KUKA KRL data list: A_154.dat

&ACCESS RVP
&REL 89
&PARAM EDITMASK = *
&PARAM TEMPLATE = C:\KRC\Roboter\Template\vorgabe
&PARAM DISKPATH = KRC:\R1\Program\T
DEFDAT  A_154
;FOLD EXTERNAL DECLARATIONS;%{PE}%MKUKATPBASIS,%CEXT,%VCOMMON,%P
;FOLD BASISTECH EXT;%{PE}%MKUKATPBASIS,%CEXT,%VEXT,%P
EXT  BAS (BAS_COMMAND  :IN,REAL  :IN )
DECL INT SUCCESS
;ENDFOLD (BASISTECH EXT)
;FOLD USER EXT;%{E}%MKUKATPUSER,%CEXT,%VEXT,%P
;Make your modifications here

;ENDFOLD (USER EXT)
;ENDFOLD (EXTERNAL DECLARATIONS)


DECL E6POS POS2={X 0.0,Y 0.0,Z 0.0,A 0.0,B 0.0,C 0.0}
DECL FDAT FS2={TOOL_NO 1,BASE_NO 1,IPO_FRAME #BASE,POINT2[] " ",TQ_STATE FALSE}
DECL LDAT LL2={VEL 0.0450000,ACC 100.000,APO_DIST 55.0000,APO_FAC 50.0000,AXIS_VEL 100.000,AXIS_ACC 100.000,ORI_TYP #VAR,CIRC_TYP #BASE,JERK_FAC 50.0000,GEAR_JERK 50.0000,EXAX_IGN 0}
DECL E6POS XP1={X 1765.00,Y -1.00106798E-34,Z 1784.00,A 0.0,B 90.0000,C 3.24968692E-36,S 2,T 34,E1 0.0,E2 0.0,E3 0.0,E4 0.0,E5 0.0,E6 0.0}
DECL FDAT FP1={TOOL_NO 1,BASE_NO 0,IPO_FRAME #BASE,POINT2[] " "}
DECL PDAT PPDAT1={VEL 100.000,ACC 100.000,APO_DIST 100.000,APO_MODE #CPTP,GEAR_JERK 100.000,EXAX_IGN 0}
DECL MODULEPARAM_T LAST_TP_PARAMS={PARAMS[] "Kuka.PointName=P6; Kuka.FrameData.base_no=0; Kuka.FrameData.tool_no=1; Kuka.FrameData.ipo_frame=#BASE; Kuka.isglobalpoint=False; Kuka.MoveDataPtpName=PDAT6; Kuka.MovementDataPdat.apo_mode=#CPTP; Kuka.MovementDataPdat.apo_dist=100; Kuka.MovementData.vel=100; Kuka.MovementData.acc=100; Kuka.MovementData.gear_jerk=100; Kuka.MovementData.exax_ign=0; Kuka.VelocityPtp=100; Kuka.BlendingEnabled=False; Kuka.CurrentCDSetIndex=0          "}
DECL E6POS XP2={X 1765.00,Y -1.00106855E-34,Z 1784.00,A 0.0,B 90.0000,C 3.24968513E-36,S 2,T 34,E1 0.0,E2 0.0,E3 0.0,E4 0.0,E5 0.0,E6 0.0}
DECL FDAT FP2={TOOL_NO 1,BASE_NO 0,IPO_FRAME #BASE,POINT2[] " "}
DECL PDAT PPDAT2={VEL 100.000,ACC 100.000,APO_DIST 100.000,APO_MODE #CPTP,GEAR_JERK 100.000,EXAX_IGN 0}
DECL E6POS XP3={X 1765.00,Y -1.00106752E-34,Z 1784.00,A 0.0,B 90.0000,C 3.24968513E-36,S 2,T 2,E1 0.0,E2 0.0,E3 0.0,E4 0.0,E5 0.0,E6 0.0}
DECL FDAT FP3={TOOL_NO 1,BASE_NO 0,IPO_FRAME #BASE,POINT2[] " "}
DECL PDAT PPDAT3={VEL 100.000,ACC 100.000,APO_DIST 100.000,APO_MODE #CPTP,GEAR_JERK 100.000,EXAX_IGN 0}
DECL E6POS XP4={X 1795.10388,Y 3.17657602E-24,Z 1784.00,A 0.0,B 90.0000,C -1.03118683E-25,S 2,T 43,E1 0.0,E2 0.0,E3 0.0,E4 0.0,E5 0.0,E6 0.0}
DECL FDAT FP4={TOOL_NO 1,BASE_NO 0,IPO_FRAME #BASE,POINT2[] " "}
DECL PDAT PPDAT4={VEL 100.000,ACC 100.000,APO_DIST 100.000,APO_MODE #CPTP,GEAR_JERK 100.000,EXAX_IGN 0}
DECL E6POS XP5={X 1795.10388,Y 0.186128840,Z 1783.99988,A 0.0,B 90.0000458,C -1.50988681E-05,S 2,T 35,E1 0.0,E2 0.0,E3 0.0,E4 0.0,E5 0.0,E6 0.0}
DECL FDAT FP5={TOOL_NO 1,BASE_NO 0,IPO_FRAME #BASE,POINT2[] " "}
DECL PDAT PPDAT5={VEL 100.000,ACC 100.000,APO_DIST 100.000,APO_MODE #CPTP,GEAR_JERK 100.000,EXAX_IGN 0}
DECL E6POS XP6={X 1795.10388,Y 0.588755548,Z 1783.99939,A 0.0,B 90.0001526,C -4.70552841E-05,S 2,T 35,E1 0.0,E2 0.0,E3 0.0,E4 0.0,E5 0.0,E6 0.0}
DECL FDAT FP6={TOOL_NO 1,BASE_NO 0,IPO_FRAME #BASE,POINT2[] " "}
DECL PDAT PPDAT6={VEL 100.000,ACC 100.000,APO_DIST 100.000,APO_MODE #CPTP,GEAR_JERK 100.000,EXAX_IGN 0}
ENDDAT
